(*

## Short summary
This interface provides assert statements for 32 bit ``DATE``  

.. <legal notes>

legal notes
=================
| SPDX-FileCopyrightText: © 2022 ekvip automation GmbH <info@ekvip.de>
| SPDX-License-Identifier: Apache-2.0
| For details check: Apache-2.0_

.. _Apache-2.0: https://www.apache.org/licenses/LICENSE-2.0

.. </legal notes>



*)

INTERFACE I32BitDateAssertions EXTENDS __SYSTEM.IQueryInterface

(*

## Short summary
This assertion method checks if the current value is equal to the expected value

.. <legal notes>

legal notes
=================
| SPDX-FileCopyrightText: © 2022 ekvip automation GmbH <info@ekvip.de>
| SPDX-License-Identifier: Apache-2.0
| For details check: Apache-2.0_

.. _Apache-2.0: https://www.apache.org/licenses/LICENSE-2.0

.. </legal notes>



*)

METHOD valueIsEqualTo
VAR_INPUT
	(* current value to check *)
	currentValue	:DATE;
	(* expected value to compare *)
	expectedValue	:DATE;
	(* message if the assertion is false *)
	message			:AssertMessage;
END_VAR
END_METHOD

(*

## Short summary
This assertion method checks if the current value is greater than the less value

.. <legal notes>

legal notes
=================
| SPDX-FileCopyrightText: © 2022 ekvip automation GmbH <info@ekvip.de>
| SPDX-License-Identifier: Apache-2.0
| For details check: Apache-2.0_

.. _Apache-2.0: https://www.apache.org/licenses/LICENSE-2.0

.. </legal notes>



*)

METHOD valueIsGreaterThan
VAR_INPUT
	(* current value to check *)
	currentValue	:DATE;
	(* less than lower limit *)
	lessValue		:DATE;
	(* message if the assertion is false *)
	message			:AssertMessage;
END_VAR
END_METHOD

(*

## Short summary
This assertion method checks if the current value is inside a limit

**Attention:** 
	limits are included: ``valueIsInRangeOf(date#1970-01-01, date#1970-01-01, date#1970-01-01)``
	is a true assertion

.. <legal notes>

legal notes
=================
| SPDX-FileCopyrightText: © 2022 ekvip automation GmbH <info@ekvip.de>
| SPDX-License-Identifier: Apache-2.0
| For details check: Apache-2.0_

.. _Apache-2.0: https://www.apache.org/licenses/LICENSE-2.0

.. </legal notes>



*)

METHOD valueIsInRangeOf
VAR_INPUT
	(* lower limit for the current value *)
	lowerLimit		:DATE;
	(* current value to check *)
	currentValue	:DATE;
	(* upper limit for the current value *)
	upperLimit		:DATE;
	(* message if the assertion is false *)
	message			:AssertMessage;
END_VAR
END_METHOD

(*

## Short summary
This assertion method checks if the current value is less than the greater value

.. <legal notes>

legal notes
=================
| SPDX-FileCopyrightText: © 2022 ekvip automation GmbH <info@ekvip.de>
| SPDX-License-Identifier: Apache-2.0
| For details check: Apache-2.0_

.. _Apache-2.0: https://www.apache.org/licenses/LICENSE-2.0

.. </legal notes>



*)

METHOD valueIsLessThan
VAR_INPUT
	(* current value to check *)
	currentValue	:DATE;
	(* greater than upper limit *)
	greaterValue	:DATE;
	(* message if the assertion is false *)
	message			:AssertMessage;
END_VAR
END_METHOD

(*

## Short summary
This assertion method checks if the current value is less than or equal to the maximum value

.. <legal notes>

legal notes
=================
| SPDX-FileCopyrightText: © 2022 ekvip automation GmbH <info@ekvip.de>
| SPDX-License-Identifier: Apache-2.0
| For details check: Apache-2.0_

.. _Apache-2.0: https://www.apache.org/licenses/LICENSE-2.0

.. </legal notes>



*)

METHOD valueIsMax
VAR_INPUT
	(* current value to check *)
	currentValue	:DATE;
	(* upper limit for the current value *)
	maximumValue	:DATE;
	(* message if the assertion is false *)
	message			:AssertMessage;
END_VAR
END_METHOD

(*

## Short summary
This assertion method checks if the current value is greater than or equal to the minimum value

.. <legal notes>

legal notes
=================
| SPDX-FileCopyrightText: © 2022 ekvip automation GmbH <info@ekvip.de>
| SPDX-License-Identifier: Apache-2.0
| For details check: Apache-2.0_

.. _Apache-2.0: https://www.apache.org/licenses/LICENSE-2.0

.. </legal notes>



*)

METHOD valueIsMin
VAR_INPUT
	(* current value to check *)
	currentValue	:DATE;
	(* lower limit for the current value *)
	minimumValue	:DATE;
	(* message if the assertion is false *)
	message			:AssertMessage;
END_VAR
END_METHOD

(*

## Short summary
This assertion method checks if the current value is not equal to the unexpected value

.. <legal notes>

legal notes
=================
| SPDX-FileCopyrightText: © 2022 ekvip automation GmbH <info@ekvip.de>
| SPDX-License-Identifier: Apache-2.0
| For details check: Apache-2.0_

.. _Apache-2.0: https://www.apache.org/licenses/LICENSE-2.0

.. </legal notes>



*)

METHOD valueIsNotEqualTo
VAR_INPUT
	(* current value to check *)
	currentValue	:DATE;
	(* unexpected value to compare *)
	unexpectedValue	:DATE;
	(* message if the assertion is false *)
	message			:AssertMessage;
END_VAR
END_METHOD

END_INTERFACE

(* stored: Version 1.1.0.1, ProductVersion 3.1.4026.8
   Itf I32BitDateAssertions: Id {2846bf71-d164-458f-bf8b-40af46183213}
   Method valueIsEqualTo: Id {6d761238-3432-4234-bc20-ac03147c8e66}
   Method valueIsGreaterThan: Id {94ae5495-b78e-46dd-ba18-897362f1c61e}
   Method valueIsInRangeOf: Id {e2d6cb8d-7fe7-45c4-b9fa-c57137fd4467}
   Method valueIsLessThan: Id {538394ac-5352-47bb-8a26-4c4f1200e2fb}
   Method valueIsMax: Id {63174092-0bc5-4c5f-b087-91ebd91bfcf4}
   Method valueIsMin: Id {82505e97-4ef5-443e-a387-2550466af349}
   Method valueIsNotEqualTo: Id {8b0e3056-1359-45b8-8dd8-1bbb6386473d} *)
